// TIA Portal V20 export
TYPE "LER_typeCommunicationData_S2I"
// stored: Access Published
   STRUCT
      UnitStatus : "LER_typeCommunicationUnitStatus";
      Common : "LER_typeCommonData";
      UnitHmiData : Array[1..50] of "LER_typeUnitHmiData";
      InterfaceData : "LER_typeCommunicationInterfaceData";
   END_STRUCT;
   // // InterfaceData."Bool"[0] : Heartbeat
   // // InterfaceData."Bool"[1] : ReadyForOperation
   // // InterfaceData."Bool"[2] : ReachedHome
   // // InterfaceData."Bool"[3] : MachineInOperation
   // // InterfaceData."Bool"[4] : NoInterference
   // // InterfaceData."Bool"[10] : PartClamped
   // // InterfaceData."Bool"[11] : PartUnclamped
   // // InterfaceData."Bool"[16] : RequestClamp
   // // InterfaceData."Bool"[17] : PartOn
   // // InterfaceData."Bool"[18] : PartReady
   // // InterfaceData."Bool"[19] : LoaderInTranferArea
   // // InterfaceData."Bool"[20] : CollisionAreaOn
   // // InterfaceData."Bool"[21] : CollisionAreaOff
   // // InterfaceData."Bool"[23] : LoadComplete
   // // InterfaceData."Bool"[26] : DataCatchUp
   // // InterfaceData."Bool"[27] : DataCompareOK
   // // InterfaceData."Bool"[28] : DataDeleted
   // // InterfaceData."Bool"[32] : NG PartReady
   // // InterfaceData."Bool"[33] : NG RequestClamp
   // // InterfaceData."Bool"[34] : NG LoadComplete
   // // InterfaceData."Bool"[40] : FATMode.Apply
   // // InterfaceData."Bool"[41] : HoursTestMode.On/Off.CMD
   // // InterfaceData."Bool"[42] : CapabilityMode.On/Off.CMD
   // // InterfaceData."Bool"[48] : ReturnToHome
   // // InterfaceData."Bool"[49] : AutoStart
   // // InterfaceData."Bool"[50] : EndOfCycle
   // // InterfaceData."Bool"[51] : StopForOpenGate
   // // InterfaceData.LReal[0] : HoursTestMode_SetTime
   // // InterfaceData.LReal[1] : CapabilityCountSetValue
END_TYPE
